FUNCTION_BLOCK FB_Alimentar_SFC

VAR_INPUT
    // SFC-Flags
    SFCPause: BOOL;
    SFCReset: BOOL;
    
    // Sincronizacion
    Benido: BOOL ;
    Ejecuta: BOOL;   
 
    //AlimentadorDelante AT %I* : BOOL;
    
END_VAR
VAR_OUTPUT
    // Sincronizacion    
    Acabhe: BOOL;
    ListoKalisto: BOOL;

  //  AlimentadorAvanza AT %Q* : BOOL;
  AlimentadorAvanza : BOOL;
END_VAR
VAR  
END_VAR

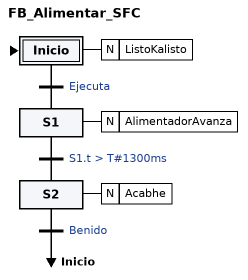
INITIAL_STEP Inicio:
    ListoKalisto(N);
END_STEP
TRANSITION FROM Inicio TO S1
    := Ejecuta;
END_TRANSITION
STEP S1:
    AlimentadorAvanza(N);
END_STEP
TRANSITION FROM S1 TO S2
    := S1.t > T#1300ms;
END_TRANSITION
STEP S2:
    Acabhe(N);
END_STEP
TRANSITION FROM S2 TO Inicio
    := Benido;
END_TRANSITION

END_FUNCTION_BLOCK

(* stored: Version 1.1.0.1, ProductVersion 3.1.4024.12
   POU FB_Alimentar_SFC: Id {e4920ed2-dd54-40ed-8583-ba2d9e57aa3e}, SpecialFunc None *)
